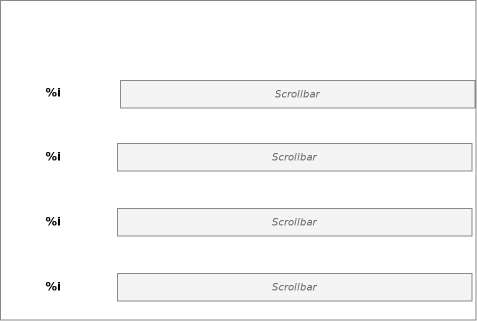
VISUALIZATION StartVisu  // 477x321
    Scrollbar (117,143 355x28)
        p1057716461: PLC_PRG.fbDMXMasterLine1.byRed
    Rectangle (10,124 87x65), "%i", text variable: PLC_PRG.fbDMXMasterLine1.byRed
    Rectangle (10,189 87x65), "%i", text variable: PLC_PRG.fbDMXMasterLine1.byGreen
    Rectangle (10,254 87x65), "%i", text variable: PLC_PRG.fbDMXMasterLine1.byBlue
    Scrollbar (117,208 355x28)
        p1057716461: PLC_PRG.fbDMXMasterLine1.byGreen
    Scrollbar (117,273 355x28)
        p1057716461: PLC_PRG.fbDMXMasterLine1.byBlue
    Scrollbar (120,80 355x28)
        p1057716461: PLC_PRG.fbDMXMasterLine1.byWhite
    Rectangle (10,60 87x65), "%i", text variable: PLC_PRG.fbDMXMasterLine1.byWhite
END_VISUALIZATION

(* stored: Version 1.1.0.1, ProductVersion 3.1.4018.5
   Visu StartVisu: Id {0b8467c5-61c6-4001-ae19-5ba3d0128d41} *)
